// TIA Portal V21 export
DATA_BLOCK "PrioritàStazioni"   // DB74
{ S7_Optimized_Access := 'TRUE' }
// stored: MemoryReserve 100
   VAR RETAIN
      K_StazioneVisualizzata { S7_SetPoint := 'True'} : Int := 16;   // K della stazione di cui intendiamo conoscere le sorgenti e le destinazioni
      K_StazioniConPriorità { S7_SetPoint := 'True'} : Array[0.."K_NumStazione"] of Int;
      K_StazioniSorgenti { S7_SetPoint := 'True'} : Array[0.."K_NumStazione"] of Int;   // Elenco delle stazioni trovate in sorgente
      K_StazioniDestinazioni { S7_SetPoint := 'True'} : Array[0.."K_NumStazione"] of Int;   // Elenco delle stazioni trovate in destinazione
      StazioniSorgenti_PrioritàHmi { S7_SetPoint := 'True'} : Array[0.."K_NumStazione"] of "Priorità";   // Soglie e isteresi indicizzate delle sorgenti
      StazioniDestinazioni_PrioritàHmi { S7_SetPoint := 'True'} : Array[0.."K_NumStazione"] of "Priorità";   // Soglie e isteresi indicizzate delle destinazioni
      Old_StazioniSorgenti_PrioritàHmi { S7_SetPoint := 'True'} : Array[0.."K_NumStazione"] of "Priorità";
      Old_StazioniDestinazioni_PrioritàHmi { S7_SetPoint := 'True'} : Array[0.."K_NumStazione"] of "Priorità";
      Old_K_StazioneVisualizzata { S7_SetPoint := 'True'} : Int := 16;
   END_VAR
BEGIN
   K_StazioniConPriorità[0] := 16;
   K_StazioniConPriorità[1] := 18;
   K_StazioniSorgenti[0] := 48;
   K_StazioniSorgenti[1] := 49;
   K_StazioniDestinazioni[0] := 1;
   K_StazioniDestinazioni[1] := 2;
END_DATA_BLOCK
